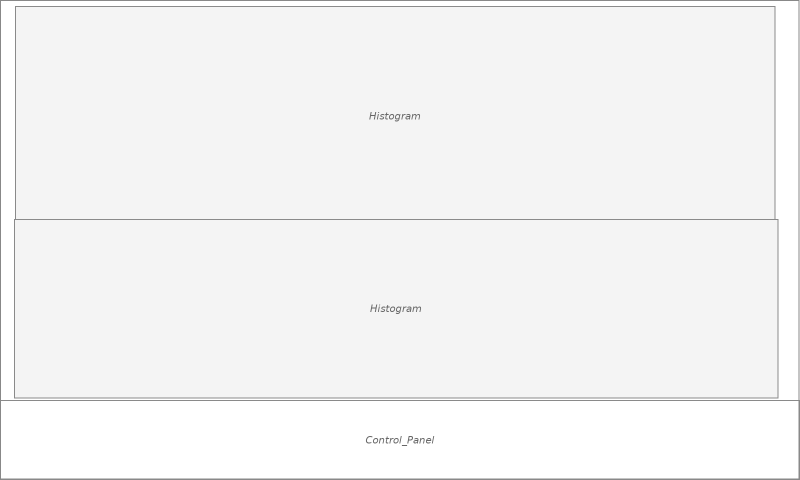
VISUALIZATION Graph  // 800x480
    Frame (0,400 800x80)
        shows Control_Panel()
    Histogram (15,6 760x220), scale format: %.0D, scale -500..500
        p518627256: Position PV, mm
        p1518820177: GVL_IO.Position_PV_mem
        p102497268: GVL_IO.Position_PV_mem
        p788070771: ARRAY [0..500] OF DINT
    Histogram (14,219 764x179), scale format: %.1f, scale 0..100
        p518627256: Motor I, Amper
        p1518820177: GVL_IO.Motor_I_mem
        p102497268: GVL_IO.Motor_I_mem
        p788070771: ARRAY [0..500] OF REAL
END_VISUALIZATION

(* stored: Version 1.1.0.1, ProductVersion 3.1.4024.13
   Visu Graph: Id {0d08c222-fbb9-47c4-9972-1f2ee75c06ca} *)
